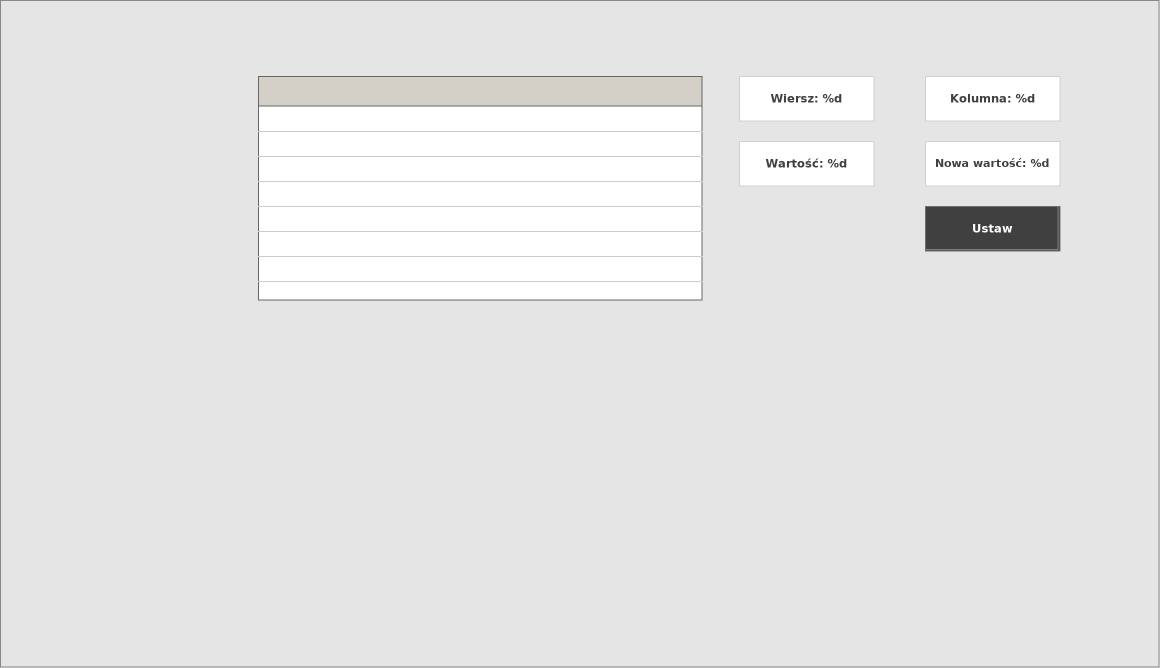
VISUALIZATION V_Table  // 1160x668
VAR_IN_OUT
	arrTable 								: ARRAY[1..10,1..10] OF INT;
	iColumn 								: INT;
	iLine 									: INT;
	iValue									: INT;
	iSetValue								: INT;
	bSet									: BOOL;
END_VAR
    Table (258,76 444x224), data array: arrTable
        p3854506369: arrTable[1,INDEX]
        p1892666644: arrTable[2,INDEX]
        p338671338: arrTable[3,INDEX]
        p2170511999: arrTable[4,INDEX]
        p3723444502: arrTable[5,INDEX]
        p1218418051: arrTable[6,INDEX]
        p746581629: arrTable[7,INDEX]
        p3104783080: arrTable[8,INDEX]
        p2501879983: arrTable[9,INDEX]
        p7306298: arrTable[10,INDEX]
        p1420305297: P_Table.iColumn
        p1137915858: P_Table.iLine
    Textfield (739,76 135x45), "Wiersz: %d", text variable: iLine
    Textfield (925,76 135x45), "Kolumna: %d", text variable: iColumn
    Textfield (739,141 135x45), "Wartość: %d", text variable: iValue
    Textfield (925,141 135x45), "Nowa wartość: %d", text variable: iSetValue
        OnMouseDown: write the text variable via Edit
    Button (925,206 135x45), "Ustaw"
        tap bSet
END_VISUALIZATION

(* stored: Version 1.1.0.1, ProductVersion 3.1.4024.3
   Visu V_Table: Id {6974c35b-4c18-49cd-aa02-d156d9e78208} *)
